{attribute 'OPC.UA.DA' := '1'}
	{attribute 'OPC.UA.DA.StructuredType' := '1'}
TYPE Breakout :
STRUCT
	RedLight	AT %Q*:BOOL; 
	AmberLight	AT %Q*:BOOL;
	GreenLight	AT %Q*:BOOL;
	BlueLight  	AT %Q*:BOOL;
	ButtonPushed AT %I*:BOOL;
END_STRUCT
END_TYPE

(* stored: Version 1.1.0.1, ProductVersion 3.1.4024.11
   DUT Breakout: Id {30c12718-b137-4546-8881-6a1889ff0049} *)
